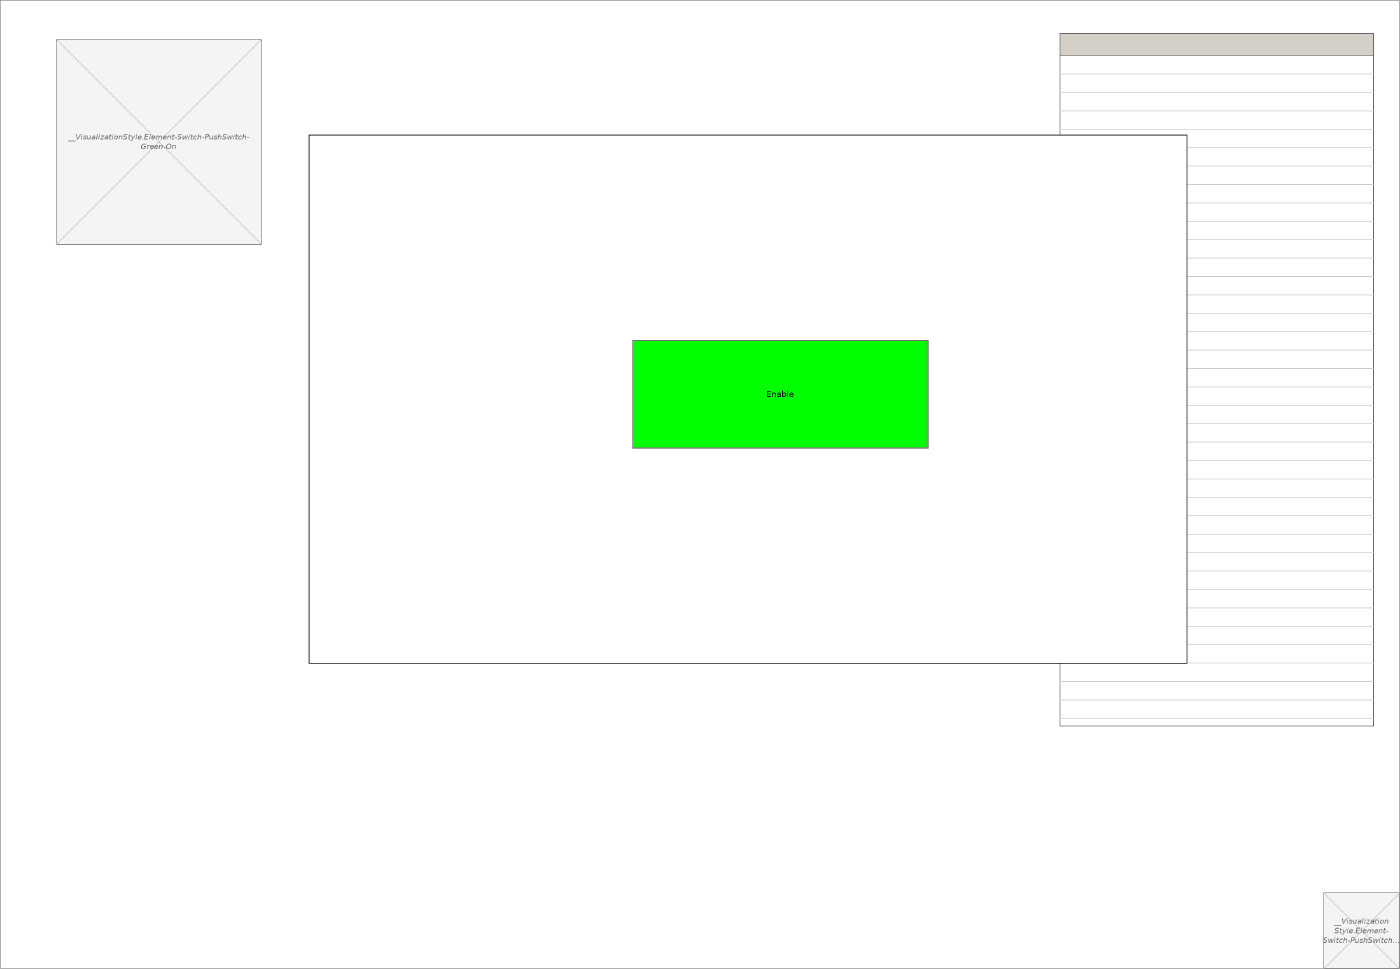
VISUALIZATION RaceControls  // 1900x1316, background image ImagePool.race-track-with-start-or-finish-line-free-vector
    Image (76,53 279x279)
        OnMouseClick: toggle MAIN.START_RACE
    Image (1796,1212 104x104)
        OnMouseClick: change screen: Settings
    Table (1438,45 426x941), data array: WinnersList.Winner_Array
        p3854506369: WinnersList.Winner_Array[INDEX]
        p2232123230: Previous Winners
        p1014161805: 10 - 1 + INT#1
    RoundedRectangle (419,183 1192x718), text variable: MAIN.cmdFB.Aborted, invisible if: MAIN.Enabled_State
    Button (858,462 402x147), "Enable", invisible if: MAIN.Enabled_State
        tap MAIN.bEnable
END_VISUALIZATION

(* stored: Version 1.1.0.1
   Visu RaceControls: Id {207ba73a-e6b6-4217-bb53-42aebb63fdee} *)
